FUNCTION_BLOCK TEMPLATE_SIFB
  (* Standard: 61499-2 *)
  (* Version 1.0, 03-07-12, GASR, Universidade do Estado de Santa Catarina *)
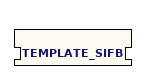
END_FUNCTION_BLOCK
